FUNCTION_BLOCK PML_Sample_Class
VAR_INPUT
END_VAR
VAR_OUTPUT
END_VAR
VAR
	stateMachine : PMLStateMachine;
	iStateMachine : IPmlStateMachine := stateMachine;
	undefined : Undefined_State(THIS, iStateMachine);
	aborting : Aborting_State(THIS, iStateMachine);
	aborted : Aborted_State(THIS, iStateMachine);
	clearing : Clearing_State(THIS, iStateMachine);
	stopped : Stopped_State(THIS, iStateMachine);
	resetting : Resetting_State_Sample(THIS, iStateMachine);
	idle : Idle_State(THIS, iStateMachine);
	starting : Starting_State_Sample(THIS, iStateMachine);
	execute : Execute_State_Sample(THIS, iStateMachine);
	iState : ITF_State := undefined;
END_VAR

iState.Cycle();
stateMachine();

METHOD SetState : BOOL
VAR_INPUT
  newState : ITF_State;
END_VAR
THIS^.iState := newState;
END_METHOD

END_FUNCTION_BLOCK

(* stored: Version 1.1.0.1, ProductVersion 3.1.4024.11
   POU PML_Sample_Class: Id {f78eb148-8bab-4ff6-9045-48ab7929f8b7}, SpecialFunc None
   Method SetState: Id {bd6b5862-4402-4e14-90a6-697d178b5813} *)
